(* IEC 61131-3 sources: F100R_S278_Temperville/MyController.device.xml.v3^/Plc Logic.plclogic.xml.v3^/Application.application.xml.v3^/04_PID/HEAT/10_Temperatura (part 3) *)

//// SUPERIORES

// Controle Resistencia 51

SR_ControleTemperatura.FbCrtlAquecimento[51](
	i_xEnable:= InterfaceHeat.P_xHabTemp51 OR xLigaDesligaSupG01,
	i_rSetPoint:= rSetPointTemperaturaSuperior[1],
	i_rProcessValue:= I_rTemperatura51,
	i_xManualMode:= ,
	i_rManualValue:= ,
	i_xAutoTune:= TEMP.xAutoTuneTemp51 OR xAutoTuneTempGeral,
	i_xHold:= ,
	i_xReset:= InterfaceHeat.xReset,
	i_stTemperatureControl:= stTemperatureControl[51],
	iq_etSelectParameterSetPID:= etSelectParameterSetPID[51],
	iq_stParameterSetsPID:= stParameterSetsPID[51],
	q_xActive=> ,
	q_xReady=> ,
	q_xError=> TEMP.xCrtlTemperatura[51],
	q_etResult=> TEMP.iCrtlTempStsTemp51,
	q_sResultMsg=> ,
	q_rAnalogOutput=> TEMP.rCrtlTempPotTemp51,
	q_xPwmOutput=> Q_xAquecimento51,
	q_xAutoTuneActive=> TEMP.xAutoTuneAtivoTemp51,
	q_etStatusAutoTune=> TEMP.iAutoTuneStsTemp51);

rPwmEntrada[51]:= TEMP.rCrtlTempPotTemp51*(rSetPorcentagemSuperior[1]/100);

PWM[51].i_stPara.tCyclTime:=T#10MS;
PWM[51].i_stPara.tPwmPeriod:=T#1000MS;
PWM[51](
	i_xEn:= 	xHabilitaBlocosControleSuperior,
	i_rIput:= 	rPwmEntrada[51],
	i_stPara:= 	,
	i_xErrRst:= xResetPid,
	q_xEn=> 	,
	q_xBusy=> 	,
	q_xPstv=> 	Q_xAquecimentoPwm51,
	q_xNgtv=> 	,
	q_xErr=> 	,
	q_uiErrId=> );

// Controle Resistencia 52

SR_ControleTemperatura.FbCrtlAquecimento[52](
	i_xEnable:= InterfaceHeat.P_xHabTemp52 OR xLigaDesligaSupG02,
	i_rSetPoint:= rSetPointTemperaturaSuperior[2],
	i_rProcessValue:= I_rTemperatura52,
	i_xManualMode:= ,
	i_rManualValue:= ,
	i_xAutoTune:= TEMP.xAutoTuneTemp52 OR xAutoTuneTempGeral,
	i_xHold:= ,
	i_xReset:= InterfaceHeat.xReset,
	i_stTemperatureControl:= stTemperatureControl[52],
	iq_etSelectParameterSetPID:= etSelectParameterSetPID[52],
	iq_stParameterSetsPID:= stParameterSetsPID[52],
	q_xActive=> ,
	q_xReady=> ,
	q_xError=> TEMP.xCrtlTemperatura[52],
	q_etResult=> TEMP.iCrtlTempStsTemp52,
	q_sResultMsg=> ,
	q_rAnalogOutput=> TEMP.rCrtlTempPotTemp52,
	q_xPwmOutput=> Q_xAquecimento52,
	q_xAutoTuneActive=> TEMP.xAutoTuneAtivoTemp52,
	q_etStatusAutoTune=> TEMP.iAutoTuneStsTemp52);

rPwmEntrada[52]:= TEMP.rCrtlTempPotTemp52*(rSetPorcentagemSuperior[2]/100);

PWM[52].i_stPara.tCyclTime:=T#10MS;
PWM[52].i_stPara.tPwmPeriod:=T#1000MS;
PWM[52](
	i_xEn:= 	xHabilitaBlocosControleSuperior,
	i_rIput:= 	rPwmEntrada[52],
	i_stPara:= 	,
	i_xErrRst:= xResetPid,
	q_xEn=> 	,
	q_xBusy=> 	,
	q_xPstv=> 	Q_xAquecimentoPwm52,
	q_xNgtv=> 	,
	q_xErr=> 	,
	q_uiErrId=> );

// Controle Resistencia 53

SR_ControleTemperatura.FbCrtlAquecimento[53](
	i_xEnable:= InterfaceHeat.P_xHabTemp53 OR xLigaDesligaSupG01,
	i_rSetPoint:= rSetPointTemperaturaSuperior[3],
	i_rProcessValue:= I_rTemperatura53,
	i_xManualMode:= ,
	i_rManualValue:= ,
	i_xAutoTune:= TEMP.xAutoTuneTemp53 OR xAutoTuneTempGeral,
	i_xHold:= ,
	i_xReset:= InterfaceHeat.xReset,
	i_stTemperatureControl:= stTemperatureControl[53],
	iq_etSelectParameterSetPID:= etSelectParameterSetPID[53],
	iq_stParameterSetsPID:= stParameterSetsPID[53],
	q_xActive=> ,
	q_xReady=> ,
	q_xError=> TEMP.xCrtlTemperatura[53],
	q_etResult=> TEMP.iCrtlTempStsTemp53,
	q_sResultMsg=> ,
	q_rAnalogOutput=> TEMP.rCrtlTempPotTemp53,
	q_xPwmOutput=> Q_xAquecimento53,
	q_xAutoTuneActive=> TEMP.xAutoTuneAtivoTemp53,
	q_etStatusAutoTune=> TEMP.iAutoTuneStsTemp53);

rPwmEntrada[53]:= TEMP.rCrtlTempPotTemp53*(rSetPorcentagemSuperior[3]/100);

PWM[53].i_stPara.tCyclTime:=T#10MS;
PWM[53].i_stPara.tPwmPeriod:=T#1000MS;
PWM[53](
	i_xEn:= 	xHabilitaBlocosControleSuperior,
	i_rIput:= 	rPwmEntrada[53],
	i_stPara:= 	,
	i_xErrRst:= xResetPid,
	q_xEn=> 	,
	q_xBusy=> 	,
	q_xPstv=> 	Q_xAquecimentoPwm53,
	q_xNgtv=> 	,
	q_xErr=> 	,
	q_uiErrId=> );

// Controle Resistencia 54

SR_ControleTemperatura.FbCrtlAquecimento[54](
	i_xEnable:= InterfaceHeat.P_xHabTemp54 OR xLigaDesligaSupG02,
	i_rSetPoint:= rSetPointTemperaturaSuperior[4],
	i_rProcessValue:= I_rTemperatura54,
	i_xManualMode:= ,
	i_rManualValue:= ,
	i_xAutoTune:= TEMP.xAutoTuneTemp54 OR xAutoTuneTempGeral,
	i_xHold:= ,
	i_xReset:= InterfaceHeat.xReset,
	i_stTemperatureControl:= stTemperatureControl[54],
	iq_etSelectParameterSetPID:= etSelectParameterSetPID[54],
	iq_stParameterSetsPID:= stParameterSetsPID[54],
	q_xActive=> ,
	q_xReady=> ,
	q_xError=> TEMP.xCrtlTemperatura[54],
	q_etResult=> TEMP.iCrtlTempStsTemp54,
	q_sResultMsg=> ,
	q_rAnalogOutput=> TEMP.rCrtlTempPotTemp54,
	q_xPwmOutput=> Q_xAquecimento54,
	q_xAutoTuneActive=> TEMP.xAutoTuneAtivoTemp54,
	q_etStatusAutoTune=> TEMP.iAutoTuneStsTemp54);

rPwmEntrada[54]:= TEMP.rCrtlTempPotTemp54*(rSetPorcentagemSuperior[4]/100);

PWM[54].i_stPara.tCyclTime:=T#10MS;
PWM[54].i_stPara.tPwmPeriod:=T#1000MS;
PWM[54](
	i_xEn:= 	xHabilitaBlocosControleSuperior,
	i_rIput:= 	rPwmEntrada[54],
	i_stPara:= 	,
	i_xErrRst:= xResetPid,
	q_xEn=> 	,
	q_xBusy=> 	,
	q_xPstv=> 	Q_xAquecimentoPwm54,
	q_xNgtv=> 	,
	q_xErr=> 	,
	q_uiErrId=> );

// Controle Resistencia 55

SR_ControleTemperatura.FbCrtlAquecimento[55](
	i_xEnable:= InterfaceHeat.P_xHabTemp55 OR xLigaDesligaSupG01,
	i_rSetPoint:= rSetPointTemperaturaSuperior[5],
	i_rProcessValue:= I_rTemperatura55,
	i_xManualMode:= ,
	i_rManualValue:= ,
	i_xAutoTune:= TEMP.xAutoTuneTemp55 OR xAutoTuneTempGeral,
	i_xHold:= ,
	i_xReset:= InterfaceHeat.xReset,
	i_stTemperatureControl:= stTemperatureControl[55],
	iq_etSelectParameterSetPID:= etSelectParameterSetPID[55],
	iq_stParameterSetsPID:= stParameterSetsPID[55],
	q_xActive=> ,
	q_xReady=> ,
	q_xError=> TEMP.xCrtlTemperatura[55],
	q_etResult=> TEMP.iCrtlTempStsTemp55,
	q_sResultMsg=> ,
	q_rAnalogOutput=> TEMP.rCrtlTempPotTemp55,
	q_xPwmOutput=> Q_xAquecimento55,
	q_xAutoTuneActive=> TEMP.xAutoTuneAtivoTemp55,
	q_etStatusAutoTune=> TEMP.iAutoTuneStsTemp55);

rPwmEntrada[55]:= TEMP.rCrtlTempPotTemp55*(rSetPorcentagemSuperior[5]/100);

PWM[55].i_stPara.tCyclTime:=T#10MS;
PWM[55].i_stPara.tPwmPeriod:=T#1000MS;
PWM[55](
	i_xEn:= 	xHabilitaBlocosControleSuperior,
	i_rIput:= 	rPwmEntrada[55],
	i_stPara:= 	,
	i_xErrRst:= xResetPid,
	q_xEn=> 	,
	q_xBusy=> 	,
	q_xPstv=> 	Q_xAquecimentoPwm55,
	q_xNgtv=> 	,
	q_xErr=> 	,
	q_uiErrId=> );

// Controle Resistencia 56

SR_ControleTemperatura.FbCrtlAquecimento[56](
	i_xEnable:= InterfaceHeat.P_xHabTemp56 OR xLigaDesligaSupG02,
	i_rSetPoint:= rSetPointTemperaturaSuperior[6],
	i_rProcessValue:= I_rTemperatura56,
	i_xManualMode:= ,
	i_rManualValue:= ,
	i_xAutoTune:= TEMP.xAutoTuneTemp56 OR xAutoTuneTempGeral,
	i_xHold:= ,
	i_xReset:= InterfaceHeat.xReset,
	i_stTemperatureControl:= stTemperatureControl[56],
	iq_etSelectParameterSetPID:= etSelectParameterSetPID[56],
	iq_stParameterSetsPID:= stParameterSetsPID[56],
	q_xActive=> ,
	q_xReady=> ,
	q_xError=> TEMP.xCrtlTemperatura[56],
	q_etResult=> TEMP.iCrtlTempStsTemp56,
	q_sResultMsg=> ,
	q_rAnalogOutput=> TEMP.rCrtlTempPotTemp56,
	q_xPwmOutput=> Q_xAquecimento56,
	q_xAutoTuneActive=> TEMP.xAutoTuneAtivoTemp56,
	q_etStatusAutoTune=> TEMP.iAutoTuneStsTemp56);

rPwmEntrada[56]:= TEMP.rCrtlTempPotTemp56*(rSetPorcentagemSuperior[6]/100);

PWM[56].i_stPara.tCyclTime:=T#10MS;
PWM[56].i_stPara.tPwmPeriod:=T#1000MS;
PWM[56](
	i_xEn:= 	xHabilitaBlocosControleSuperior,
	i_rIput:= 	rPwmEntrada[56],
	i_stPara:= 	,
	i_xErrRst:= xResetPid,
	q_xEn=> 	,
	q_xBusy=> 	,
	q_xPstv=> 	Q_xAquecimentoPwm56,
	q_xNgtv=> 	,
	q_xErr=> 	,
	q_uiErrId=> );

// Controle Resistencia 57

SR_ControleTemperatura.FbCrtlAquecimento[57](
	i_xEnable:= InterfaceHeat.P_xHabTemp57 OR xLigaDesligaSupG01,
	i_rSetPoint:= rSetPointTemperaturaSuperior[7],
	i_rProcessValue:= I_rTemperatura57,
	i_xManualMode:= ,
	i_rManualValue:= ,
	i_xAutoTune:= TEMP.xAutoTuneTemp57 OR xAutoTuneTempGeral,
	i_xHold:= ,
	i_xReset:= InterfaceHeat.xReset,
	i_stTemperatureControl:= stTemperatureControl[57],
	iq_etSelectParameterSetPID:= etSelectParameterSetPID[57],
	iq_stParameterSetsPID:= stParameterSetsPID[57],
	q_xActive=> ,
	q_xReady=> ,
	q_xError=> TEMP.xCrtlTemperatura[57],
	q_etResult=> TEMP.iCrtlTempStsTemp57,
	q_sResultMsg=> ,
	q_rAnalogOutput=> TEMP.rCrtlTempPotTemp57,
	q_xPwmOutput=> Q_xAquecimento57,
	q_xAutoTuneActive=> TEMP.xAutoTuneAtivoTemp57,
	q_etStatusAutoTune=> TEMP.iAutoTuneStsTemp57);

rPwmEntrada[57]:= TEMP.rCrtlTempPotTemp57*(rSetPorcentagemSuperior[7]/100);

PWM[57].i_stPara.tCyclTime:=T#10MS;
PWM[57].i_stPara.tPwmPeriod:=T#1000MS;
PWM[57](
	i_xEn:= 	xHabilitaBlocosControleSuperior,
	i_rIput:= 	rPwmEntrada[57],
	i_stPara:= 	,
	i_xErrRst:= xResetPid,
	q_xEn=> 	,
	q_xBusy=> 	,
	q_xPstv=> 	Q_xAquecimentoPwm57,
	q_xNgtv=> 	,
	q_xErr=> 	,
	q_uiErrId=> );

	// Controle Resistencia 58

SR_ControleTemperatura.FbCrtlAquecimento[58](
	i_xEnable:= InterfaceHeat.P_xHabTemp58 OR xLigaDesligaSupG02,
	i_rSetPoint:= rSetPointTemperaturaSuperior[8],
	i_rProcessValue:= I_rTemperatura58,
	i_xManualMode:= ,
	i_rManualValue:= ,
	i_xAutoTune:= TEMP.xAutoTuneTemp58 OR xAutoTuneTempGeral,
	i_xHold:= ,
	i_xReset:= InterfaceHeat.xReset,
	i_stTemperatureControl:= stTemperatureControl[58],
	iq_etSelectParameterSetPID:= etSelectParameterSetPID[58],
	iq_stParameterSetsPID:= stParameterSetsPID[58],
	q_xActive=> ,
	q_xReady=> ,
	q_xError=> TEMP.xCrtlTemperatura[58],
	q_etResult=> TEMP.iCrtlTempStsTemp58,
	q_sResultMsg=> ,
	q_rAnalogOutput=> TEMP.rCrtlTempPotTemp58,
	q_xPwmOutput=> Q_xAquecimento58,
	q_xAutoTuneActive=> TEMP.xAutoTuneAtivoTemp58,
	q_etStatusAutoTune=> TEMP.iAutoTuneStsTemp58);

rPwmEntrada[58]:= TEMP.rCrtlTempPotTemp58*(rSetPorcentagemSuperior[8]/100);

PWM[58].i_stPara.tCyclTime:=T#10MS;
PWM[58].i_stPara.tPwmPeriod:=T#1000MS;
PWM[58](
	i_xEn:= 	xHabilitaBlocosControleSuperior,
	i_rIput:= 	rPwmEntrada[58],
	i_stPara:= 	,
	i_xErrRst:= xResetPid,
	q_xEn=> 	,
	q_xBusy=> 	,
	q_xPstv=> 	Q_xAquecimentoPwm58,
	q_xNgtv=> 	,
	q_xErr=> 	,
	q_uiErrId=> );

	// Controle Resistencia 59

SR_ControleTemperatura.FbCrtlAquecimento[59](
	i_xEnable:= InterfaceHeat.P_xHabTemp59 OR xLigaDesligaSupG01,
	i_rSetPoint:= rSetPointTemperaturaSuperior[9],
	i_rProcessValue:= I_rTemperatura59,
	i_xManualMode:= ,
	i_rManualValue:= ,
	i_xAutoTune:= TEMP.xAutoTuneTemp59 OR xAutoTuneTempGeral,
	i_xHold:= ,
	i_xReset:= InterfaceHeat.xReset,
	i_stTemperatureControl:= stTemperatureControl[59],
	iq_etSelectParameterSetPID:= etSelectParameterSetPID[59],
	iq_stParameterSetsPID:= stParameterSetsPID[59],
	q_xActive=> ,
	q_xReady=> ,
	q_xError=> TEMP.xCrtlTemperatura[59],
	q_etResult=> TEMP.iCrtlTempStsTemp59,
	q_sResultMsg=> ,
	q_rAnalogOutput=> TEMP.rCrtlTempPotTemp59,
	q_xPwmOutput=> Q_xAquecimento59,
	q_xAutoTuneActive=> TEMP.xAutoTuneAtivoTemp59,
	q_etStatusAutoTune=> TEMP.iAutoTuneStsTemp59);

rPwmEntrada[59]:= TEMP.rCrtlTempPotTemp59*(rSetPorcentagemSuperior[9]/100);

PWM[59].i_stPara.tCyclTime:=T#10MS;
PWM[59].i_stPara.tPwmPeriod:=T#1000MS;
PWM[59](
	i_xEn:= 	xHabilitaBlocosControleSuperior,
	i_rIput:= 	rPwmEntrada[59],
	i_stPara:= 	,
	i_xErrRst:= xResetPid,
	q_xEn=> 	,
	q_xBusy=> 	,
	q_xPstv=> 	Q_xAquecimentoPwm59,
	q_xNgtv=> 	,
	q_xErr=> 	,
	q_uiErrId=> );

	// Controle Resistencia 60

SR_ControleTemperatura.FbCrtlAquecimento[60](
	i_xEnable:= InterfaceHeat.P_xHabTemp60 OR xLigaDesligaSupG02,
	i_rSetPoint:= rSetPointTemperaturaSuperior[10],
	i_rProcessValue:= I_rTemperatura60,
	i_xManualMode:= ,
	i_rManualValue:= ,
	i_xAutoTune:= TEMP.xAutoTuneTemp60 OR xAutoTuneTempGeral,
	i_xHold:= ,
	i_xReset:= InterfaceHeat.xReset,
	i_stTemperatureControl:= stTemperatureControl[60],
	iq_etSelectParameterSetPID:= etSelectParameterSetPID[60],
	iq_stParameterSetsPID:= stParameterSetsPID[60],
	q_xActive=> ,
	q_xReady=> ,
	q_xError=> TEMP.xCrtlTemperatura[60],
	q_etResult=> TEMP.iCrtlTempStsTemp60,
	q_sResultMsg=> ,
	q_rAnalogOutput=> TEMP.rCrtlTempPotTemp60,
	q_xPwmOutput=> Q_xAquecimento60,
	q_xAutoTuneActive=> TEMP.xAutoTuneAtivoTemp60,
	q_etStatusAutoTune=> TEMP.iAutoTuneStsTemp60);

rPwmEntrada[60]:= TEMP.rCrtlTempPotTemp60*(rSetPorcentagemSuperior[10]/100);

PWM[60].i_stPara.tCyclTime:=T#10MS;
PWM[60].i_stPara.tPwmPeriod:=T#1000MS;
PWM[60](
	i_xEn:= 	xHabilitaBlocosControleSuperior,
	i_rIput:= 	rPwmEntrada[60],
	i_stPara:= 	,
	i_xErrRst:= xResetPid,
	q_xEn=> 	,
	q_xBusy=> 	,
	q_xPstv=> 	Q_xAquecimentoPwm60,
	q_xNgtv=> 	,
	q_xErr=> 	,
	q_uiErrId=> );

// Controle Resistencia 61

SR_ControleTemperatura.FbCrtlAquecimento[61](
	i_xEnable:= InterfaceHeat.P_xHabTemp61 OR xLigaDesligaSupG02,
	i_rSetPoint:= rSetPointTemperaturaSuperior[11],
	i_rProcessValue:= I_rTemperatura61,
	i_xManualMode:= ,
	i_rManualValue:= ,
	i_xAutoTune:= TEMP.xAutoTuneTemp61 OR xAutoTuneTempGeral,
	i_xHold:= ,
	i_xReset:= InterfaceHeat.xReset,
	i_stTemperatureControl:= stTemperatureControl[61],
	iq_etSelectParameterSetPID:= etSelectParameterSetPID[61],
	iq_stParameterSetsPID:= stParameterSetsPID[61],
	q_xActive=> ,
	q_xReady=> ,
	q_xError=> TEMP.xCrtlTemperatura[61],
	q_etResult=> TEMP.iCrtlTempStsTemp61,
	q_sResultMsg=> ,
	q_rAnalogOutput=> TEMP.rCrtlTempPotTemp61,
	q_xPwmOutput=> Q_xAquecimento61,
	q_xAutoTuneActive=> TEMP.xAutoTuneAtivoTemp61,
	q_etStatusAutoTune=> TEMP.iAutoTuneStsTemp61);

rPwmEntrada[61]:= TEMP.rCrtlTempPotTemp6*(rSetPorcentagemSuperior[11]/100);

PWM[61].i_stPara.tCyclTime:=T#10MS;
PWM[61].i_stPara.tPwmPeriod:=T#1000MS;
PWM[61](
	i_xEn:= 	xHabilitaBlocosControleSuperior,
	i_rIput:= 	rPwmEntrada[61],
	i_stPara:= 	,
	i_xErrRst:= xResetPid,
	q_xEn=> 	,
	q_xBusy=> 	,
	q_xPstv=> 	Q_xAquecimentoPwm61,
	q_xNgtv=> 	,
	q_xErr=> 	,
	q_uiErrId=> );

// Controle Resistencia 62

SR_ControleTemperatura.FbCrtlAquecimento[62](
	i_xEnable:= InterfaceHeat.P_xHabTemp62 OR xLigaDesligaSupG01,
	i_rSetPoint:= rSetPointTemperaturaSuperior[12],
	i_rProcessValue:= I_rTemperatura62,
	i_xManualMode:= ,
	i_rManualValue:= ,
	i_xAutoTune:= TEMP.xAutoTuneTemp62 OR xAutoTuneTempGeral,
	i_xHold:= ,
	i_xReset:= InterfaceHeat.xReset,
	i_stTemperatureControl:= stTemperatureControl[62],
	iq_etSelectParameterSetPID:= etSelectParameterSetPID[62],
	iq_stParameterSetsPID:= stParameterSetsPID[62],
	q_xActive=> ,
	q_xReady=> ,
	q_xError=> TEMP.xCrtlTemperatura[62],
	q_etResult=> TEMP.iCrtlTempStsTemp62,
	q_sResultMsg=> ,
	q_rAnalogOutput=> TEMP.rCrtlTempPotTemp62,
	q_xPwmOutput=> Q_xAquecimento62,
	q_xAutoTuneActive=> TEMP.xAutoTuneAtivoTemp62,
	q_etStatusAutoTune=> TEMP.iAutoTuneStsTemp62);

rPwmEntrada[62]:= TEMP.rCrtlTempPotTemp62*(rSetPorcentagemSuperior[12]/100);

PWM[62].i_stPara.tCyclTime:=T#10MS;
PWM[62].i_stPara.tPwmPeriod:=T#1000MS;
PWM[62](
	i_xEn:= 	xHabilitaBlocosControleSuperior,
	i_rIput:= 	rPwmEntrada[62],
	i_stPara:= 	,
	i_xErrRst:= xResetPid,
	q_xEn=> 	,
	q_xBusy=> 	,
	q_xPstv=> 	Q_xAquecimentoPwm62,
	q_xNgtv=> 	,
	q_xErr=> 	,
	q_uiErrId=> );

// Controle Resistencia 63

SR_ControleTemperatura.FbCrtlAquecimento[63](
	i_xEnable:= InterfaceHeat.P_xHabTemp63 OR xLigaDesligaSupG02,
	i_rSetPoint:= rSetPointTemperaturaSuperior[13],
	i_rProcessValue:= I_rTemperatura63,
	i_xManualMode:= ,
	i_rManualValue:= ,
	i_xAutoTune:= TEMP.xAutoTuneTemp63 OR xAutoTuneTempGeral,
	i_xHold:= ,
	i_xReset:= InterfaceHeat.xReset,
	i_stTemperatureControl:= stTemperatureControl[63],
	iq_etSelectParameterSetPID:= etSelectParameterSetPID[63],
	iq_stParameterSetsPID:= stParameterSetsPID[63],
	q_xActive=> ,
	q_xReady=> ,
	q_xError=> TEMP.xCrtlTemperatura[63],
	q_etResult=> TEMP.iCrtlTempStsTemp63,
	q_sResultMsg=> ,
	q_rAnalogOutput=> TEMP.rCrtlTempPotTemp63,
	q_xPwmOutput=> Q_xAquecimento63,
	q_xAutoTuneActive=> TEMP.xAutoTuneAtivoTemp63,
	q_etStatusAutoTune=> TEMP.iAutoTuneStsTemp63);

rPwmEntrada[63]:= TEMP.rCrtlTempPotTemp63*(rSetPorcentagemSuperior[13]/100);

PWM[63].i_stPara.tCyclTime:=T#10MS;
PWM[63].i_stPara.tPwmPeriod:=T#1000MS;
PWM[63](
	i_xEn:= 	xHabilitaBlocosControleSuperior,
	i_rIput:= 	rPwmEntrada[63],
	i_stPara:= 	,
	i_xErrRst:= xResetPid,
	q_xEn=> 	,
	q_xBusy=> 	,
	q_xPstv=> 	Q_xAquecimentoPwm63,
	q_xNgtv=> 	,
	q_xErr=> 	,
	q_uiErrId=> );

// Controle Resistencia 64

SR_ControleTemperatura.FbCrtlAquecimento[64](
	i_xEnable:= InterfaceHeat.P_xHabTemp64 OR xLigaDesligaSupG01,
	i_rSetPoint:= rSetPointTemperaturaSuperior[14],
	i_rProcessValue:= I_rTemperatura64,
	i_xManualMode:= ,
	i_rManualValue:= ,
	i_xAutoTune:= TEMP.xAutoTuneTemp64 OR xAutoTuneTempGeral,
	i_xHold:= ,
	i_xReset:= InterfaceHeat.xReset,
	i_stTemperatureControl:= stTemperatureControl[64],
	iq_etSelectParameterSetPID:= etSelectParameterSetPID[64],
	iq_stParameterSetsPID:= stParameterSetsPID[64],
	q_xActive=> ,
	q_xReady=> ,
	q_xError=> TEMP.xCrtlTemperatura[64],
	q_etResult=> TEMP.iCrtlTempStsTemp64,
	q_sResultMsg=> ,
	q_rAnalogOutput=> TEMP.rCrtlTempPotTemp64,
	q_xPwmOutput=> Q_xAquecimento64,
	q_xAutoTuneActive=> TEMP.xAutoTuneAtivoTemp64,
	q_etStatusAutoTune=> TEMP.iAutoTuneStsTemp64);

rPwmEntrada[64]:= TEMP.rCrtlTempPotTemp64*(rSetPorcentagemSuperior[14]/100);

PWM[64].i_stPara.tCyclTime:=T#10MS;
PWM[64].i_stPara.tPwmPeriod:=T#1000MS;
PWM[64](
	i_xEn:= 	xHabilitaBlocosControleSuperior,
	i_rIput:= 	rPwmEntrada[64],
	i_stPara:= 	,
	i_xErrRst:= xResetPid,
	q_xEn=> 	,
	q_xBusy=> 	,
	q_xPstv=> 	Q_xAquecimentoPwm64,
	q_xNgtv=> 	,
	q_xErr=> 	,
	q_uiErrId=> );

// Controle Resistencia 65

SR_ControleTemperatura.FbCrtlAquecimento[65](
	i_xEnable:= InterfaceHeat.P_xHabTemp65 OR xLigaDesligaSupG02,
	i_rSetPoint:= rSetPointTemperaturaSuperior[15],
	i_rProcessValue:= I_rTemperatura65,
	i_xManualMode:= ,
	i_rManualValue:= ,
	i_xAutoTune:= TEMP.xAutoTuneTemp65 OR xAutoTuneTempGeral,
	i_xHold:= ,
	i_xReset:= InterfaceHeat.xReset,
	i_stTemperatureControl:= stTemperatureControl[65],
	iq_etSelectParameterSetPID:= etSelectParameterSetPID[65],
	iq_stParameterSetsPID:= stParameterSetsPID[65],
	q_xActive=> ,
	q_xReady=> ,
	q_xError=> TEMP.xCrtlTemperatura[65],
	q_etResult=> TEMP.iCrtlTempStsTemp65,
	q_sResultMsg=> ,
	q_rAnalogOutput=> TEMP.rCrtlTempPotTemp65,
	q_xPwmOutput=> Q_xAquecimento65,
	q_xAutoTuneActive=> TEMP.xAutoTuneAtivoTemp65,
	q_etStatusAutoTune=> TEMP.iAutoTuneStsTemp65);

rPwmEntrada[65]:= TEMP.rCrtlTempPotTemp65*(rSetPorcentagemSuperior[15]/100);

PWM[65].i_stPara.tCyclTime:=T#10MS;
PWM[65].i_stPara.tPwmPeriod:=T#1000MS;
PWM[65](
	i_xEn:= 	xHabilitaBlocosControleSuperior,
	i_rIput:= 	rPwmEntrada[65],
	i_stPara:= 	,
	i_xErrRst:= xResetPid,
	q_xEn=> 	,
	q_xBusy=> 	,
	q_xPstv=> 	Q_xAquecimentoPwm65,
	q_xNgtv=> 	,
	q_xErr=> 	,
	q_uiErrId=> );

// Controle Resistencia 66

SR_ControleTemperatura.FbCrtlAquecimento[66](
	i_xEnable:= InterfaceHeat.P_xHabTemp66 OR xLigaDesligaSupG01,
	i_rSetPoint:= rSetPointTemperaturaSuperior[16],
	i_rProcessValue:= I_rTemperatura66,
	i_xManualMode:= ,
	i_rManualValue:= ,
	i_xAutoTune:= TEMP.xAutoTuneTemp66 OR xAutoTuneTempGeral,
	i_xHold:= ,
	i_xReset:= InterfaceHeat.xReset,
	i_stTemperatureControl:= stTemperatureControl[66],
	iq_etSelectParameterSetPID:= etSelectParameterSetPID[66],
	iq_stParameterSetsPID:= stParameterSetsPID[66],
	q_xActive=> ,
	q_xReady=> ,
	q_xError=> TEMP.xCrtlTemperatura[66],
	q_etResult=> TEMP.iCrtlTempStsTemp66,
	q_sResultMsg=> ,
	q_rAnalogOutput=> TEMP.rCrtlTempPotTemp66,
	q_xPwmOutput=> Q_xAquecimento66,
	q_xAutoTuneActive=> TEMP.xAutoTuneAtivoTemp66,
	q_etStatusAutoTune=> TEMP.iAutoTuneStsTemp66);

rPwmEntrada[66]:= TEMP.rCrtlTempPotTemp66*(rSetPorcentagemSuperior[16]/100);

PWM[66].i_stPara.tCyclTime:=T#10MS;
PWM[66].i_stPara.tPwmPeriod:=T#1000MS;
PWM[66](
	i_xEn:= 	xHabilitaBlocosControleSuperior,
	i_rIput:= 	rPwmEntrada[66],
	i_stPara:= 	,
	i_xErrRst:= xResetPid,
	q_xEn=> 	,
	q_xBusy=> 	,
	q_xPstv=> 	Q_xAquecimentoPwm66,
	q_xNgtv=> 	,
	q_xErr=> 	,
	q_uiErrId=> );

// Controle Resistencia 67

SR_ControleTemperatura.FbCrtlAquecimento[67](
	i_xEnable:= InterfaceHeat.P_xHabTemp67 OR xLigaDesligaSupG02,
	i_rSetPoint:= rSetPointTemperaturaSuperior[17],
	i_rProcessValue:= I_rTemperatura67,
	i_xManualMode:= ,
	i_rManualValue:= ,
	i_xAutoTune:= TEMP.xAutoTuneTemp67 OR xAutoTuneTempGeral,
	i_xHold:= ,
	i_xReset:= InterfaceHeat.xReset,
	i_stTemperatureControl:= stTemperatureControl[67],
	iq_etSelectParameterSetPID:= etSelectParameterSetPID[67],
	iq_stParameterSetsPID:= stParameterSetsPID[67],
	q_xActive=> ,
	q_xReady=> ,
	q_xError=> TEMP.xCrtlTemperatura[67],
	q_etResult=> TEMP.iCrtlTempStsTemp67,
	q_sResultMsg=> ,
	q_rAnalogOutput=> TEMP.rCrtlTempPotTemp67,
	q_xPwmOutput=> Q_xAquecimento67,
	q_xAutoTuneActive=> TEMP.xAutoTuneAtivoTemp67,
	q_etStatusAutoTune=> TEMP.iAutoTuneStsTemp67);

rPwmEntrada[67]:= TEMP.rCrtlTempPotTemp67*(rSetPorcentagemSuperior[17]/100);

PWM[67].i_stPara.tCyclTime:=T#10MS;
PWM[67].i_stPara.tPwmPeriod:=T#1000MS;
PWM[67](
	i_xEn:= 	xHabilitaBlocosControleSuperior,
	i_rIput:= 	rPwmEntrada[67],
	i_stPara:= 	,
	i_xErrRst:= xResetPid,
	q_xEn=> 	,
	q_xBusy=> 	,
	q_xPstv=> 	Q_xAquecimentoPwm67,
	q_xNgtv=> 	,
	q_xErr=> 	,
	q_uiErrId=> );

	// Controle Resistencia 68

SR_ControleTemperatura.FbCrtlAquecimento[68](
	i_xEnable:= InterfaceHeat.P_xHabTemp68 OR xLigaDesligaSupG01,
	i_rSetPoint:= rSetPointTemperaturaSuperior[18],
	i_rProcessValue:= I_rTemperatura68,
	i_xManualMode:= ,
	i_rManualValue:= ,
	i_xAutoTune:= TEMP.xAutoTuneTemp68 OR xAutoTuneTempGeral,
	i_xHold:= ,
	i_xReset:= InterfaceHeat.xReset,
	i_stTemperatureControl:= stTemperatureControl[68],
	iq_etSelectParameterSetPID:= etSelectParameterSetPID[68],
	iq_stParameterSetsPID:= stParameterSetsPID[68],
	q_xActive=> ,
	q_xReady=> ,
	q_xError=> TEMP.xCrtlTemperatura[68],
	q_etResult=> TEMP.iCrtlTempStsTemp68,
	q_sResultMsg=> ,
	q_rAnalogOutput=> TEMP.rCrtlTempPotTemp68,
	q_xPwmOutput=> Q_xAquecimento68,
	q_xAutoTuneActive=> TEMP.xAutoTuneAtivoTemp68,
	q_etStatusAutoTune=> TEMP.iAutoTuneStsTemp68);

rPwmEntrada[68]:= TEMP.rCrtlTempPotTemp68*(rSetPorcentagemSuperior[18]/100);

PWM[68].i_stPara.tCyclTime:=T#10MS;
PWM[68].i_stPara.tPwmPeriod:=T#1000MS;
PWM[68](
	i_xEn:= 	xHabilitaBlocosControleSuperior,
	i_rIput:= 	rPwmEntrada[68],
	i_stPara:= 	,
	i_xErrRst:= xResetPid,
	q_xEn=> 	,
	q_xBusy=> 	,
	q_xPstv=> 	Q_xAquecimentoPwm68,
	q_xNgtv=> 	,
	q_xErr=> 	,
	q_uiErrId=> );

	// Controle Resistencia 69

SR_ControleTemperatura.FbCrtlAquecimento[69](
	i_xEnable:= InterfaceHeat.P_xHabTemp69 OR xLigaDesligaSupG02,
	i_rSetPoint:= rSetPointTemperaturaSuperior[19],
	i_rProcessValue:= I_rTemperatura69,
	i_xManualMode:= ,
	i_rManualValue:= ,
	i_xAutoTune:= TEMP.xAutoTuneTemp69 OR xAutoTuneTempGeral,
	i_xHold:= ,
	i_xReset:= InterfaceHeat.xReset,
	i_stTemperatureControl:= stTemperatureControl[69],
	iq_etSelectParameterSetPID:= etSelectParameterSetPID[69],
	iq_stParameterSetsPID:= stParameterSetsPID[69],
	q_xActive=> ,
	q_xReady=> ,
	q_xError=> TEMP.xCrtlTemperatura[69],
	q_etResult=> TEMP.iCrtlTempStsTemp69,
	q_sResultMsg=> ,
	q_rAnalogOutput=> TEMP.rCrtlTempPotTemp69,
	q_xPwmOutput=> Q_xAquecimento69,
	q_xAutoTuneActive=> TEMP.xAutoTuneAtivoTemp69,
	q_etStatusAutoTune=> TEMP.iAutoTuneStsTemp69);

rPwmEntrada[69]:= TEMP.rCrtlTempPotTemp69*(rSetPorcentagemSuperior[19]/100);

PWM[69].i_stPara.tCyclTime:=T#10MS;
PWM[69].i_stPara.tPwmPeriod:=T#1000MS;
PWM[69](
	i_xEn:= 	xHabilitaBlocosControleSuperior,
	i_rIput:= 	rPwmEntrada[69],
	i_stPara:= 	,
	i_xErrRst:= xResetPid,
	q_xEn=> 	,
	q_xBusy=> 	,
	q_xPstv=> 	Q_xAquecimentoPwm69,
	q_xNgtv=> 	,
	q_xErr=> 	,
	q_uiErrId=> );

	// Controle Resistencia 70

SR_ControleTemperatura.FbCrtlAquecimento[70](
	i_xEnable:= InterfaceHeat.P_xHabTemp70 OR xLigaDesligaSupG01,
	i_rSetPoint:= rSetPointTemperaturaSuperior[20],
	i_rProcessValue:= I_rTemperatura70,
	i_xManualMode:= ,
	i_rManualValue:= ,
	i_xAutoTune:= TEMP.xAutoTuneTemp70 OR xAutoTuneTempGeral,
	i_xHold:= ,
	i_xReset:= InterfaceHeat.xReset,
	i_stTemperatureControl:= stTemperatureControl[70],
	iq_etSelectParameterSetPID:= etSelectParameterSetPID[70],
	iq_stParameterSetsPID:= stParameterSetsPID[70],
	q_xActive=> ,
	q_xReady=> ,
	q_xError=> TEMP.xCrtlTemperatura[70],
	q_etResult=> TEMP.iCrtlTempStsTemp70,
	q_sResultMsg=> ,
	q_rAnalogOutput=> TEMP.rCrtlTempPotTemp70,
	q_xPwmOutput=> Q_xAquecimento70,
	q_xAutoTuneActive=> TEMP.xAutoTuneAtivoTemp70,
	q_etStatusAutoTune=> TEMP.iAutoTuneStsTemp70);

rPwmEntrada[70]:= TEMP.rCrtlTempPotTemp70*(rSetPorcentagemSuperior[20]/100);

PWM[70].i_stPara.tCyclTime:=T#10MS;
PWM[70].i_stPara.tPwmPeriod:=T#1000MS;
PWM[70](
	i_xEn:= 	xHabilitaBlocosControleSuperior,
	i_rIput:= 	rPwmEntrada[70],
	i_stPara:= 	,
	i_xErrRst:= xResetPid,
	q_xEn=> 	,
	q_xBusy=> 	,
	q_xPstv=> 	Q_xAquecimentoPwm70,
	q_xNgtv=> 	,
	q_xErr=> 	,
	q_uiErrId=> );

// Controle Resistencia 71

SR_ControleTemperatura.FbCrtlAquecimento[71](
	i_xEnable:= InterfaceHeat.P_xHabTemp71 OR xLigaDesligaSupG01,
	i_rSetPoint:= rSetPointTemperaturaSuperior[21],
	i_rProcessValue:= I_rTemperatura71,
	i_xManualMode:= ,
	i_rManualValue:= ,
	i_xAutoTune:= TEMP.xAutoTuneTemp71 OR xAutoTuneTempGeral,
	i_xHold:= ,
	i_xReset:= InterfaceHeat.xReset,
	i_stTemperatureControl:= stTemperatureControl[71],
	iq_etSelectParameterSetPID:= etSelectParameterSetPID[71],
	iq_stParameterSetsPID:= stParameterSetsPID[71],
	q_xActive=> ,
	q_xReady=> ,
	q_xError=> TEMP.xCrtlTemperatura[71],
	q_etResult=> TEMP.iCrtlTempStsTemp71,
	q_sResultMsg=> ,
	q_rAnalogOutput=> TEMP.rCrtlTempPotTemp71,
	q_xPwmOutput=> Q_xAquecimento71,
	q_xAutoTuneActive=> TEMP.xAutoTuneAtivoTemp71,
	q_etStatusAutoTune=> TEMP.iAutoTuneStsTemp71);

rPwmEntrada[71]:= TEMP.rCrtlTempPotTemp71*(rSetPorcentagemSuperior[21]/100);

PWM[71].i_stPara.tCyclTime:=T#10MS;
PWM[71].i_stPara.tPwmPeriod:=T#1000MS;
PWM[71](
	i_xEn:= 	xHabilitaBlocosControleSuperior,
	i_rIput:= 	rPwmEntrada[71],
	i_stPara:= 	,
	i_xErrRst:= xResetPid,
	q_xEn=> 	,
	q_xBusy=> 	,
	q_xPstv=> 	Q_xAquecimentoPwm71,
	q_xNgtv=> 	,
	q_xErr=> 	,
	q_uiErrId=> );

// Controle Resistencia 72

SR_ControleTemperatura.FbCrtlAquecimento[72](
	i_xEnable:= InterfaceHeat.P_xHabTemp72 OR xLigaDesligaSupG02,
	i_rSetPoint:= rSetPointTemperaturaSuperior[22],
	i_rProcessValue:= I_rTemperatura72,
	i_xManualMode:= ,
	i_rManualValue:= ,
	i_xAutoTune:= TEMP.xAutoTuneTemp72 OR xAutoTuneTempGeral,
	i_xHold:= ,
	i_xReset:= InterfaceHeat.xReset,
	i_stTemperatureControl:= stTemperatureControl[72],
	iq_etSelectParameterSetPID:= etSelectParameterSetPID[72],
	iq_stParameterSetsPID:= stParameterSetsPID[72],
	q_xActive=> ,
	q_xReady=> ,
	q_xError=> TEMP.xCrtlTemperatura[72],
	q_etResult=> TEMP.iCrtlTempStsTemp72,
	q_sResultMsg=> ,
	q_rAnalogOutput=> TEMP.rCrtlTempPotTemp72,
	q_xPwmOutput=> Q_xAquecimento72,
	q_xAutoTuneActive=> TEMP.xAutoTuneAtivoTemp72,
	q_etStatusAutoTune=> TEMP.iAutoTuneStsTemp72);

rPwmEntrada[72]:= TEMP.rCrtlTempPotTemp72*(rSetPorcentagemSuperior[22]/100);

PWM[72].i_stPara.tCyclTime:=T#10MS;
PWM[72].i_stPara.tPwmPeriod:=T#1000MS;
PWM[72](
	i_xEn:= 	xHabilitaBlocosControleSuperior,
	i_rIput:= 	rPwmEntrada[72],
	i_stPara:= 	,
	i_xErrRst:= xResetPid,
	q_xEn=> 	,
	q_xBusy=> 	,
	q_xPstv=> 	Q_xAquecimentoPwm72,
	q_xNgtv=> 	,
	q_xErr=> 	,
	q_uiErrId=> );

// Controle Resistencia 73

SR_ControleTemperatura.FbCrtlAquecimento[73](
	i_xEnable:= InterfaceHeat.P_xHabTemp73 OR xLigaDesligaSupG01,
	i_rSetPoint:= rSetPointTemperaturaSuperior[23],
	i_rProcessValue:= I_rTemperatura73,
	i_xManualMode:= ,
	i_rManualValue:= ,
	i_xAutoTune:= TEMP.xAutoTuneTemp73 OR xAutoTuneTempGeral,
	i_xHold:= ,
	i_xReset:= InterfaceHeat.xReset,
	i_stTemperatureControl:= stTemperatureControl[73],
	iq_etSelectParameterSetPID:= etSelectParameterSetPID[73],
	iq_stParameterSetsPID:= stParameterSetsPID[73],
	q_xActive=> ,
	q_xReady=> ,
	q_xError=> TEMP.xCrtlTemperatura[73],
	q_etResult=> TEMP.iCrtlTempStsTemp73,
	q_sResultMsg=> ,
	q_rAnalogOutput=> TEMP.rCrtlTempPotTemp73,
	q_xPwmOutput=> Q_xAquecimento73,
	q_xAutoTuneActive=> TEMP.xAutoTuneAtivoTemp73,
	q_etStatusAutoTune=> TEMP.iAutoTuneStsTemp73);

rPwmEntrada[73]:= TEMP.rCrtlTempPotTemp73*(rSetPorcentagemSuperior[23]/100);

PWM[73].i_stPara.tCyclTime:=T#10MS;
PWM[73].i_stPara.tPwmPeriod:=T#1000MS;
PWM[73](
	i_xEn:= 	xHabilitaBlocosControleSuperior,
	i_rIput:= 	rPwmEntrada[73],
	i_stPara:= 	,
	i_xErrRst:= xResetPid,
	q_xEn=> 	,
	q_xBusy=> 	,
	q_xPstv=> 	Q_xAquecimentoPwm73,
	q_xNgtv=> 	,
	q_xErr=> 	,
	q_uiErrId=> );

// Controle Resistencia 74

SR_ControleTemperatura.FbCrtlAquecimento[74](
	i_xEnable:= InterfaceHeat.P_xHabTemp74 OR xLigaDesligaSupG02,
	i_rSetPoint:= rSetPointTemperaturaSuperior[24],
	i_rProcessValue:= I_rTemperatura74,
	i_xManualMode:= ,
	i_rManualValue:= ,
	i_xAutoTune:= TEMP.xAutoTuneTemp74 OR xAutoTuneTempGeral,
	i_xHold:= ,
	i_xReset:= InterfaceHeat.xReset,
	i_stTemperatureControl:= stTemperatureControl[74],
	iq_etSelectParameterSetPID:= etSelectParameterSetPID[74],
	iq_stParameterSetsPID:= stParameterSetsPID[74],
	q_xActive=> ,
	q_xReady=> ,
	q_xError=> TEMP.xCrtlTemperatura[74],
	q_etResult=> TEMP.iCrtlTempStsTemp74,
	q_sResultMsg=> ,
	q_rAnalogOutput=> TEMP.rCrtlTempPotTemp74,
	q_xPwmOutput=> Q_xAquecimento74,
	q_xAutoTuneActive=> TEMP.xAutoTuneAtivoTemp74,
	q_etStatusAutoTune=> TEMP.iAutoTuneStsTemp74);

rPwmEntrada[74]:= TEMP.rCrtlTempPotTemp74*(rSetPorcentagemSuperior[24]/100);

PWM[74].i_stPara.tCyclTime:=T#10MS;
PWM[74].i_stPara.tPwmPeriod:=T#1000MS;
PWM[74](
	i_xEn:= 	xHabilitaBlocosControleSuperior,
	i_rIput:= 	rPwmEntrada[74],
	i_stPara:= 	,
	i_xErrRst:= xResetPid,
	q_xEn=> 	,
	q_xBusy=> 	,
	q_xPstv=> 	Q_xAquecimentoPwm74,
	q_xNgtv=> 	,
	q_xErr=> 	,
	q_uiErrId=> );

// Controle Resistencia 75

FbAqueceRampa[75](
	iTermopar:= TermoparLogicoSuperior[25],
	rSpTemperatura:= rSetPointTemperaturaSuperior[25],
	iTempoEstab:= iTempoEstabRampa,
	xReset:= ,
	xStartRampaCiclo=> ,
	xRampaAtiva=> xRampaAqAtiva[75],
	TemperUp=> ,
	TemperDown=> ,
	rSpTemperaturaUp=> ,
	rSetTemperaturaRampa=> rSetTemperaturaRampaAq[75] );

SR_ControleTemperatura.FbCrtlAquecimento[75](
	i_xEnable:= InterfaceHeat.P_xHabTemp75 OR xLigaDesligaSupG01,
	i_rSetPoint:= rSetPointTemperaturaSuperior[25],
	i_rProcessValue:= I_rTemperatura75,
	i_xManualMode:= ,
	i_rManualValue:= ,
	i_xAutoTune:= TEMP.xAutoTuneTemp75 OR xAutoTuneTempGeral,
	i_xHold:= ,
	i_xReset:= InterfaceHeat.xReset,
	i_stTemperatureControl:= stTemperatureControl[75],
	iq_etSelectParameterSetPID:= etSelectParameterSetPID[75],
	iq_stParameterSetsPID:= stParameterSetsPID[75],
	q_xActive=> ,
	q_xReady=> ,
	q_xError=> TEMP.xCrtlTemperatura[75],
	q_etResult=> TEMP.iCrtlTempStsTemp75,
	q_sResultMsg=> ,
	q_rAnalogOutput=> TEMP.rCrtlTempPotTemp75,
	q_xPwmOutput=> Q_xAquecimento75,
	q_xAutoTuneActive=> TEMP.xAutoTuneAtivoTemp75,
	q_etStatusAutoTune=> TEMP.iAutoTuneStsTemp75);

rPwmEntrada[75]:= TEMP.rCrtlTempPotTemp75*(rSetPorcentagemSuperior[25]/100);

PWM[75].i_stPara.tCyclTime:=T#10MS;
PWM[75].i_stPara.tPwmPeriod:=T#1000MS;
PWM[75](
	i_xEn:= 	xHabilitaBlocosControleSuperior,
	i_rIput:= 	rPwmEntrada[75],
	i_stPara:= 	,
	i_xErrRst:= xResetPid,
	q_xEn=> 	,
	q_xBusy=> 	,
	q_xPstv=> 	Q_xAquecimentoPwm75,
	q_xNgtv=> 	,
	q_xErr=> 	,
	q_uiErrId=> );

	(*IF xRampaAqAtiva[75] THEN
		xReleSsrSuperior[25]:=Q_xAquecimento75;
	ELSE
		xReleSsrSuperior[25]:=Q_xAquecimentoPwm75;
	END_IF*)

// Controle Resistencia 76

SR_ControleTemperatura.FbCrtlAquecimento[76](
	i_xEnable:= InterfaceHeat.P_xHabTemp76 OR xLigaDesligaSupG02,
	i_rSetPoint:= rSetPointTemperaturaSuperior[26],
	i_rProcessValue:= I_rTemperatura76,
	i_xManualMode:= ,
	i_rManualValue:= ,
	i_xAutoTune:= TEMP.xAutoTuneTemp76 OR xAutoTuneTempGeral,
	i_xHold:= ,
	i_xReset:= InterfaceHeat.xReset,
	i_stTemperatureControl:= stTemperatureControl[76],
	iq_etSelectParameterSetPID:= etSelectParameterSetPID[76],
	iq_stParameterSetsPID:= stParameterSetsPID[76],
	q_xActive=> ,
	q_xReady=> ,
	q_xError=> TEMP.xCrtlTemperatura[76],
	q_etResult=> TEMP.iCrtlTempStsTemp76,
	q_sResultMsg=> ,
	q_rAnalogOutput=> TEMP.rCrtlTempPotTemp76,
	q_xPwmOutput=> Q_xAquecimento76,
	q_xAutoTuneActive=> TEMP.xAutoTuneAtivoTemp76,
	q_etStatusAutoTune=> TEMP.iAutoTuneStsTemp76);

rPwmEntrada[76]:= TEMP.rCrtlTempPotTemp76*(rSetPorcentagemSuperior[26]/100);

PWM[76].i_stPara.tCyclTime:=T#10MS;
PWM[76].i_stPara.tPwmPeriod:=T#1000MS;
PWM[76](
	i_xEn:= 	xHabilitaBlocosControleSuperior,
	i_rIput:= 	rPwmEntrada[76],
	i_stPara:= 	,
	i_xErrRst:= xResetPid,
	q_xEn=> 	,
	q_xBusy=> 	,
	q_xPstv=> 	Q_xAquecimentoPwm76,
	q_xNgtv=> 	,
	q_xErr=> 	,
	q_uiErrId=> );

// Controle Resistencia 77

SR_ControleTemperatura.FbCrtlAquecimento[77](
	i_xEnable:= InterfaceHeat.P_xHabTemp77 OR xLigaDesligaSupG01,
	i_rSetPoint:= rSetPointTemperaturaSuperior[27],
	i_rProcessValue:= I_rTemperatura77,
	i_xManualMode:= ,
	i_rManualValue:= ,
	i_xAutoTune:= TEMP.xAutoTuneTemp77 OR xAutoTuneTempGeral,
	i_xHold:= ,
	i_xReset:= InterfaceHeat.xReset,
	i_stTemperatureControl:= stTemperatureControl[77],
	iq_etSelectParameterSetPID:= etSelectParameterSetPID[77],
	iq_stParameterSetsPID:= stParameterSetsPID[77],
	q_xActive=> ,
	q_xReady=> ,
	q_xError=> TEMP.xCrtlTemperatura[77],
	q_etResult=> TEMP.iCrtlTempStsTemp77,
	q_sResultMsg=> ,
	q_rAnalogOutput=> TEMP.rCrtlTempPotTemp77,
	q_xPwmOutput=> Q_xAquecimento77,
	q_xAutoTuneActive=> TEMP.xAutoTuneAtivoTemp77,
	q_etStatusAutoTune=> TEMP.iAutoTuneStsTemp77);

rPwmEntrada[77]:= TEMP.rCrtlTempPotTemp77*(rSetPorcentagemSuperior[27]/100);

PWM[77].i_stPara.tCyclTime:=T#10MS;
PWM[77].i_stPara.tPwmPeriod:=T#1000MS;
PWM[77](
	i_xEn:= 	xHabilitaBlocosControleSuperior,
	i_rIput:= 	rPwmEntrada[77],
	i_stPara:= 	,
	i_xErrRst:= xResetPid,
	q_xEn=> 	,
	q_xBusy=> 	,
	q_xPstv=> 	Q_xAquecimentoPwm77,
	q_xNgtv=> 	,
	q_xErr=> 	,
	q_uiErrId=> );

	// Controle Resistencia 78

SR_ControleTemperatura.FbCrtlAquecimento[78](
	i_xEnable:= InterfaceHeat.P_xHabTemp78 OR xLigaDesligaSupG02,
	i_rSetPoint:= rSetPointTemperaturaSuperior[28],
	i_rProcessValue:= I_rTemperatura78,
	i_xManualMode:= ,
	i_rManualValue:= ,
	i_xAutoTune:= TEMP.xAutoTuneTemp78 OR xAutoTuneTempGeral,
	i_xHold:= ,
	i_xReset:= InterfaceHeat.xReset,
	i_stTemperatureControl:= stTemperatureControl[78],
	iq_etSelectParameterSetPID:= etSelectParameterSetPID[78],
	iq_stParameterSetsPID:= stParameterSetsPID[78],
	q_xActive=> ,
	q_xReady=> ,
	q_xError=> TEMP.xCrtlTemperatura[78],
	q_etResult=> TEMP.iCrtlTempStsTemp78,
	q_sResultMsg=> ,
	q_rAnalogOutput=> TEMP.rCrtlTempPotTemp78,
	q_xPwmOutput=> Q_xAquecimento78,
	q_xAutoTuneActive=> TEMP.xAutoTuneAtivoTemp78,
	q_etStatusAutoTune=> TEMP.iAutoTuneStsTemp78);

	rPwmEntrada[78]:= TEMP.rCrtlTempPotTemp78*(rSetPorcentagemSuperior[28]/100);

PWM[78].i_stPara.tCyclTime:=T#10MS;
PWM[78].i_stPara.tPwmPeriod:=T#1000MS;
PWM[78](
	i_xEn:= 	xHabilitaBlocosControleSuperior,
	i_rIput:= 	rPwmEntrada[78],
	i_stPara:= 	,
	i_xErrRst:= xResetPid,
	q_xEn=> 	,
	q_xBusy=> 	,
	q_xPstv=> 	Q_xAquecimentoPwm78,
	q_xNgtv=> 	,
	q_xErr=> 	,
	q_uiErrId=> );

// Controle Resistencia 79

SR_ControleTemperatura.FbCrtlAquecimento[79](
	i_xEnable:= InterfaceHeat.P_xHabTemp79 OR xLigaDesligaSupG01,
	i_rSetPoint:= rSetPointTemperaturaSuperior[29],
	i_rProcessValue:= I_rTemperatura79,
	i_xManualMode:= ,
	i_rManualValue:= ,
	i_xAutoTune:= TEMP.xAutoTuneTemp79 OR xAutoTuneTempGeral,
	i_xHold:= ,
	i_xReset:= InterfaceHeat.xReset,
	i_stTemperatureControl:= stTemperatureControl[79],
	iq_etSelectParameterSetPID:= etSelectParameterSetPID[79],
	iq_stParameterSetsPID:= stParameterSetsPID[79],
	q_xActive=> ,
	q_xReady=> ,
	q_xError=> TEMP.xCrtlTemperatura[79],
	q_etResult=> TEMP.iCrtlTempStsTemp79,
	q_sResultMsg=> ,
	q_rAnalogOutput=> TEMP.rCrtlTempPotTemp79,
	q_xPwmOutput=> Q_xAquecimento79,
	q_xAutoTuneActive=> TEMP.xAutoTuneAtivoTemp79,
	q_etStatusAutoTune=> TEMP.iAutoTuneStsTemp79);

	rPwmEntrada[79]:= TEMP.rCrtlTempPotTemp79*(rSetPorcentagemSuperior[29]/100);

PWM[79].i_stPara.tCyclTime:=T#10MS;
PWM[79].i_stPara.tPwmPeriod:=T#1000MS;
PWM[79](
	i_xEn:= 	xHabilitaBlocosControleSuperior,
	i_rIput:= 	rPwmEntrada[79],
	i_stPara:= 	,
	i_xErrRst:= xResetPid,
	q_xEn=> 	,
	q_xBusy=> 	,
	q_xPstv=> 	Q_xAquecimentoPwm79,
	q_xNgtv=> 	,
	q_xErr=> 	,
	q_uiErrId=> );

// Controle Resistencia 80

SR_ControleTemperatura.FbCrtlAquecimento[80](
	i_xEnable:= InterfaceHeat.P_xHabTemp80 OR xLigaDesligaSupG02,
	i_rSetPoint:= rSetPointTemperaturaSuperior[30],
	i_rProcessValue:= I_rTemperatura80,
	i_xManualMode:= ,
	i_rManualValue:= ,
	i_xAutoTune:= TEMP.xAutoTuneTemp80 OR xAutoTuneTempGeral,
	i_xHold:= ,
	i_xReset:= InterfaceHeat.xReset,
	i_stTemperatureControl:= stTemperatureControl[80],
	iq_etSelectParameterSetPID:= etSelectParameterSetPID[80],
	iq_stParameterSetsPID:= stParameterSetsPID[80],
	q_xActive=> ,
	q_xReady=> ,
	q_xError=> TEMP.xCrtlTemperatura[80],
	q_etResult=> TEMP.iCrtlTempStsTemp80,
	q_sResultMsg=> ,
	q_rAnalogOutput=> TEMP.rCrtlTempPotTemp80,
	q_xPwmOutput=> Q_xAquecimento80,
	q_xAutoTuneActive=> TEMP.xAutoTuneAtivoTemp80,
	q_etStatusAutoTune=> TEMP.iAutoTuneStsTemp80);

rPwmEntrada[80]:= TEMP.rCrtlTempPotTemp80*(rSetPorcentagemSuperior[30]/100);

PWM[80].i_stPara.tCyclTime:=T#10MS;
PWM[80].i_stPara.tPwmPeriod:=T#1000MS;
PWM[80](
	i_xEn:= 	xHabilitaBlocosControleSuperior,
	i_rIput:= 	rPwmEntrada[80],
	i_stPara:= 	,
	i_xErrRst:= xResetPid,
	q_xEn=> 	,
	q_xBusy=> 	,
	q_xPstv=> 	Q_xAquecimentoPwm80,
	q_xNgtv=> 	,
	q_xErr=> 	,
	q_uiErrId=> );

// Controle Resistencia 81

SR_ControleTemperatura.FbCrtlAquecimento[81](
	i_xEnable:= InterfaceHeat.P_xHabTemp81 OR xLigaDesligaSupG02,
	i_rSetPoint:= rSetPointTemperaturaSuperior[31],
	i_rProcessValue:= I_rTemperatura81,
	i_xManualMode:= ,
	i_rManualValue:= ,
	i_xAutoTune:= TEMP.xAutoTuneTemp81 OR xAutoTuneTempGeral,
	i_xHold:= ,
	i_xReset:= InterfaceHeat.xReset,
	i_stTemperatureControl:= stTemperatureControl[81],
	iq_etSelectParameterSetPID:= etSelectParameterSetPID[81],
	iq_stParameterSetsPID:= stParameterSetsPID[81],
	q_xActive=> ,
	q_xReady=> ,
	q_xError=> TEMP.xCrtlTemperatura[81],
	q_etResult=> TEMP.iCrtlTempStsTemp81,
	q_sResultMsg=> ,
	q_rAnalogOutput=> TEMP.rCrtlTempPotTemp81,
	q_xPwmOutput=> Q_xAquecimento81,
	q_xAutoTuneActive=> TEMP.xAutoTuneAtivoTemp81,
	q_etStatusAutoTune=> TEMP.iAutoTuneStsTemp81);

rPwmEntrada[81]:= TEMP.rCrtlTempPotTemp81*(rSetPorcentagemSuperior[31]/100);

PWM[81].i_stPara.tCyclTime:=T#10MS;
PWM[81].i_stPara.tPwmPeriod:=T#1000MS;
PWM[81](
	i_xEn:= 	xHabilitaBlocosControleSuperior,
	i_rIput:= 	rPwmEntrada[81],
	i_stPara:= 	,
	i_xErrRst:= xResetPid,
	q_xEn=> 	,
	q_xBusy=> 	,
	q_xPstv=> 	Q_xAquecimentoPwm81,
	q_xNgtv=> 	,
	q_xErr=> 	,
	q_uiErrId=> );

// Controle Resistencia 82

SR_ControleTemperatura.FbCrtlAquecimento[82](
	i_xEnable:= InterfaceHeat.P_xHabTemp82 OR xLigaDesligaSupG01,
	i_rSetPoint:= rSetPointTemperaturaSuperior[32],
	i_rProcessValue:= I_rTemperatura82,
	i_xManualMode:= ,
	i_rManualValue:= ,
	i_xAutoTune:= TEMP.xAutoTuneTemp82 OR xAutoTuneTempGeral,
	i_xHold:= ,
	i_xReset:= InterfaceHeat.xReset,
	i_stTemperatureControl:= stTemperatureControl[82],
	iq_etSelectParameterSetPID:= etSelectParameterSetPID[82],
	iq_stParameterSetsPID:= stParameterSetsPID[82],
	q_xActive=> ,
	q_xReady=> ,
	q_xError=> TEMP.xCrtlTemperatura[82],
	q_etResult=> TEMP.iCrtlTempStsTemp82,
	q_sResultMsg=> ,
	q_rAnalogOutput=> TEMP.rCrtlTempPotTemp82,
	q_xPwmOutput=> Q_xAquecimento82,
	q_xAutoTuneActive=> TEMP.xAutoTuneAtivoTemp82,
	q_etStatusAutoTune=> TEMP.iAutoTuneStsTemp82);

rPwmEntrada[82]:= TEMP.rCrtlTempPotTemp82*(rSetPorcentagemSuperior[32]/100);

PWM[82].i_stPara.tCyclTime:=T#10MS;
PWM[82].i_stPara.tPwmPeriod:=T#1000MS;
PWM[82](
	i_xEn:= 	xHabilitaBlocosControleSuperior,
	i_rIput:= 	rPwmEntrada[82],
	i_stPara:= 	,
	i_xErrRst:= xResetPid,
	q_xEn=> 	,
	q_xBusy=> 	,
	q_xPstv=> 	Q_xAquecimentoPwm82,
	q_xNgtv=> 	,
	q_xErr=> 	,
	q_uiErrId=> );

// Controle Resistencia 83

SR_ControleTemperatura.FbCrtlAquecimento[83](
	i_xEnable:= InterfaceHeat.P_xHabTemp83 OR xLigaDesligaSupG02,
	i_rSetPoint:= rSetPointTemperaturaSuperior[33],
	i_rProcessValue:= I_rTemperatura83,
	i_xManualMode:= ,
	i_rManualValue:= ,
	i_xAutoTune:= TEMP.xAutoTuneTemp83 OR xAutoTuneTempGeral,
	i_xHold:= ,
	i_xReset:= InterfaceHeat.xReset,
	i_stTemperatureControl:= stTemperatureControl[83],
	iq_etSelectParameterSetPID:= etSelectParameterSetPID[83],
	iq_stParameterSetsPID:= stParameterSetsPID[83],
	q_xActive=> ,
	q_xReady=> ,
	q_xError=> TEMP.xCrtlTemperatura[83],
	q_etResult=> TEMP.iCrtlTempStsTemp83,
	q_sResultMsg=> ,
	q_rAnalogOutput=> TEMP.rCrtlTempPotTemp83,
	q_xPwmOutput=> Q_xAquecimento83,
	q_xAutoTuneActive=> TEMP.xAutoTuneAtivoTemp83,
	q_etStatusAutoTune=> TEMP.iAutoTuneStsTemp83);

rPwmEntrada[83]:= TEMP.rCrtlTempPotTemp83*(rSetPorcentagemSuperior[33]/100);

PWM[83].i_stPara.tCyclTime:=T#10MS;
PWM[83].i_stPara.tPwmPeriod:=T#1000MS;
PWM[83](
	i_xEn:= 	xHabilitaBlocosControleSuperior,
	i_rIput:= 	rPwmEntrada[83],
	i_stPara:= 	,
	i_xErrRst:= xResetPid,
	q_xEn=> 	,
	q_xBusy=> 	,
	q_xPstv=> 	Q_xAquecimentoPwm83,
	q_xNgtv=> 	,
	q_xErr=> 	,
	q_uiErrId=> );

// Controle Resistencia 84

SR_ControleTemperatura.FbCrtlAquecimento[84](
	i_xEnable:= InterfaceHeat.P_xHabTemp84 OR xLigaDesligaSupG01,
	i_rSetPoint:= rSetPointTemperaturaSuperior[34],
	i_rProcessValue:= I_rTemperatura84,
	i_xManualMode:= ,
	i_rManualValue:= ,
	i_xAutoTune:= TEMP.xAutoTuneTemp84 OR xAutoTuneTempGeral,
	i_xHold:= ,
	i_xReset:= InterfaceHeat.xReset,
	i_stTemperatureControl:= stTemperatureControl[84],
	iq_etSelectParameterSetPID:= etSelectParameterSetPID[84],
	iq_stParameterSetsPID:= stParameterSetsPID[84],
	q_xActive=> ,
	q_xReady=> ,
	q_xError=> TEMP.xCrtlTemperatura[84],
	q_etResult=> TEMP.iCrtlTempStsTemp84,
	q_sResultMsg=> ,
	q_rAnalogOutput=> TEMP.rCrtlTempPotTemp84,
	q_xPwmOutput=> Q_xAquecimento84,
	q_xAutoTuneActive=> TEMP.xAutoTuneAtivoTemp84,
	q_etStatusAutoTune=> TEMP.iAutoTuneStsTemp84);

rPwmEntrada[84]:= TEMP.rCrtlTempPotTemp84*(rSetPorcentagemSuperior[34]/100);

PWM[84].i_stPara.tCyclTime:=T#10MS;
PWM[84].i_stPara.tPwmPeriod:=T#1000MS;
PWM[84](
	i_xEn:= 	xHabilitaBlocosControleSuperior,
	i_rIput:= 	rPwmEntrada[84],
	i_stPara:= 	,
	i_xErrRst:= xResetPid,
	q_xEn=> 	,
	q_xBusy=> 	,
	q_xPstv=> 	Q_xAquecimentoPwm84,
	q_xNgtv=> 	,
	q_xErr=> 	,
	q_uiErrId=> );

// Controle Resistencia 85

SR_ControleTemperatura.FbCrtlAquecimento[85](
	i_xEnable:= InterfaceHeat.P_xHabTemp85 OR xLigaDesligaSupG02,
	i_rSetPoint:= rSetPointTemperaturaSuperior[35],
	i_rProcessValue:= I_rTemperatura85,
	i_xManualMode:= ,
	i_rManualValue:= ,
	i_xAutoTune:= TEMP.xAutoTuneTemp85 OR xAutoTuneTempGeral,
	i_xHold:= ,
	i_xReset:= InterfaceHeat.xReset,
	i_stTemperatureControl:= stTemperatureControl[85],
	iq_etSelectParameterSetPID:= etSelectParameterSetPID[85],
	iq_stParameterSetsPID:= stParameterSetsPID[85],
	q_xActive=> ,
	q_xReady=> ,
	q_xError=> TEMP.xCrtlTemperatura[85],
	q_etResult=> TEMP.iCrtlTempStsTemp85,
	q_sResultMsg=> ,
	q_rAnalogOutput=> TEMP.rCrtlTempPotTemp85,
	q_xPwmOutput=> Q_xAquecimento85,
	q_xAutoTuneActive=> TEMP.xAutoTuneAtivoTemp85,
	q_etStatusAutoTune=> TEMP.iAutoTuneStsTemp85);

rPwmEntrada[85]:= TEMP.rCrtlTempPotTemp85*(rSetPorcentagemSuperior[35]/100);

PWM[85].i_stPara.tCyclTime:=T#10MS;
PWM[85].i_stPara.tPwmPeriod:=T#1000MS;
PWM[85](
	i_xEn:= 	xHabilitaBlocosControleSuperior,
	i_rIput:= 	rPwmEntrada[85],
	i_stPara:= 	,
	i_xErrRst:= xResetPid,
	q_xEn=> 	,
	q_xBusy=> 	,
	q_xPstv=> 	Q_xAquecimentoPwm85,
	q_xNgtv=> 	,
	q_xErr=> 	,
	q_uiErrId=> );

// Controle Resistencia 86

SR_ControleTemperatura.FbCrtlAquecimento[86](
	i_xEnable:= InterfaceHeat.P_xHabTemp86 OR xLigaDesligaSupG01,
	i_rSetPoint:= rSetPointTemperaturaSuperior[36],
	i_rProcessValue:= I_rTemperatura86,
	i_xManualMode:= ,
	i_rManualValue:= ,
	i_xAutoTune:= TEMP.xAutoTuneTemp86 OR xAutoTuneTempGeral,
	i_xHold:= ,
	i_xReset:= InterfaceHeat.xReset,
	i_stTemperatureControl:= stTemperatureControl[86],
	iq_etSelectParameterSetPID:= etSelectParameterSetPID[86],
	iq_stParameterSetsPID:= stParameterSetsPID[86],
	q_xActive=> ,
	q_xReady=> ,
	q_xError=> TEMP.xCrtlTemperatura[86],
	q_etResult=> TEMP.iCrtlTempStsTemp86,
	q_sResultMsg=> ,
	q_rAnalogOutput=> TEMP.rCrtlTempPotTemp86,
	q_xPwmOutput=> Q_xAquecimento86,
	q_xAutoTuneActive=> TEMP.xAutoTuneAtivoTemp86,
	q_etStatusAutoTune=> TEMP.iAutoTuneStsTemp86);

rPwmEntrada[86]:= TEMP.rCrtlTempPotTemp86*(rSetPorcentagemSuperior[36]/100);

PWM[86].i_stPara.tCyclTime:=T#10MS;
PWM[86].i_stPara.tPwmPeriod:=T#1000MS;
PWM[86](
	i_xEn:= 	xHabilitaBlocosControleSuperior,
	i_rIput:= 	rPwmEntrada[86],
	i_stPara:= 	,
	i_xErrRst:= xResetPid,
	q_xEn=> 	,
	q_xBusy=> 	,
	q_xPstv=> 	Q_xAquecimentoPwm86,
	q_xNgtv=> 	,
	q_xErr=> 	,
	q_uiErrId=> );

// Controle Resistencia 87

SR_ControleTemperatura.FbCrtlAquecimento[87](
	i_xEnable:= InterfaceHeat.P_xHabTemp87 OR xLigaDesligaSupG02,
	i_rSetPoint:= rSetPointTemperaturaSuperior[37],
	i_rProcessValue:= I_rTemperatura87,
	i_xManualMode:= ,
	i_rManualValue:= ,
	i_xAutoTune:= TEMP.xAutoTuneTemp87 OR xAutoTuneTempGeral,
	i_xHold:= ,
	i_xReset:= InterfaceHeat.xReset,
	i_stTemperatureControl:= stTemperatureControl[87],
	iq_etSelectParameterSetPID:= etSelectParameterSetPID[87],
	iq_stParameterSetsPID:= stParameterSetsPID[87],
	q_xActive=> ,
	q_xReady=> ,
	q_xError=> TEMP.xCrtlTemperatura[87],
	q_etResult=> TEMP.iCrtlTempStsTemp87,
	q_sResultMsg=> ,
	q_rAnalogOutput=> TEMP.rCrtlTempPotTemp87,
	q_xPwmOutput=> Q_xAquecimento87,
	q_xAutoTuneActive=> TEMP.xAutoTuneAtivoTemp87,
	q_etStatusAutoTune=> TEMP.iAutoTuneStsTemp87);

	rPwmEntrada[87]:= TEMP.rCrtlTempPotTemp87*(rSetPorcentagemSuperior[37]/100);

PWM[87].i_stPara.tCyclTime:=T#10MS;
PWM[87].i_stPara.tPwmPeriod:=T#1000MS;
PWM[87](
	i_xEn:= 	xHabilitaBlocosControleSuperior,
	i_rIput:= 	rPwmEntrada[87],
	i_stPara:= 	,
	i_xErrRst:= xResetPid,
	q_xEn=> 	,
	q_xBusy=> 	,
	q_xPstv=> 	Q_xAquecimentoPwm87,
	q_xNgtv=> 	,
	q_xErr=> 	,
	q_uiErrId=> );

// Controle Resistencia 88

SR_ControleTemperatura.FbCrtlAquecimento[88](
	i_xEnable:= InterfaceHeat.P_xHabTemp88 OR xLigaDesligaSupG01,
	i_rSetPoint:= rSetPointTemperaturaSuperior[38],
	i_rProcessValue:= I_rTemperatura88,
	i_xManualMode:= ,
	i_rManualValue:= ,
	i_xAutoTune:= TEMP.xAutoTuneTemp88 OR xAutoTuneTempGeral,
	i_xHold:= ,
	i_xReset:= InterfaceHeat.xReset,
	i_stTemperatureControl:= stTemperatureControl[88],
	iq_etSelectParameterSetPID:= etSelectParameterSetPID[88],
	iq_stParameterSetsPID:= stParameterSetsPID[88],
	q_xActive=> ,
	q_xReady=> ,
	q_xError=> TEMP.xCrtlTemperatura[88],
	q_etResult=> TEMP.iCrtlTempStsTemp88,
	q_sResultMsg=> ,
	q_rAnalogOutput=> TEMP.rCrtlTempPotTemp88,
	q_xPwmOutput=> Q_xAquecimento88,
	q_xAutoTuneActive=> TEMP.xAutoTuneAtivoTemp88,
	q_etStatusAutoTune=> TEMP.iAutoTuneStsTemp88);

rPwmEntrada[88]:= TEMP.rCrtlTempPotTemp88*(rSetPorcentagemSuperior[38]/100);

PWM[88].i_stPara.tCyclTime:=T#10MS;
PWM[88].i_stPara.tPwmPeriod:=T#1000MS;
PWM[88](
	i_xEn:= 	xHabilitaBlocosControleSuperior,
	i_rIput:= 	rPwmEntrada[88],
	i_stPara:= 	,
	i_xErrRst:= xResetPid,
	q_xEn=> 	,
	q_xBusy=> 	,
	q_xPstv=> 	Q_xAquecimentoPwm88,
	q_xNgtv=> 	,
	q_xErr=> 	,
	q_uiErrId=> );

	// Controle Resistencia 89

SR_ControleTemperatura.FbCrtlAquecimento[89](
	i_xEnable:= InterfaceHeat.P_xHabTemp89 OR xLigaDesligaSupG02,
	i_rSetPoint:= rSetPointTemperaturaSuperior[39],
	i_rProcessValue:= I_rTemperatura89,
	i_xManualMode:= ,
	i_rManualValue:= ,
	i_xAutoTune:= TEMP.xAutoTuneTemp89 OR xAutoTuneTempGeral,
	i_xHold:= ,
	i_xReset:= InterfaceHeat.xReset,
	i_stTemperatureControl:= stTemperatureControl[89],
	iq_etSelectParameterSetPID:= etSelectParameterSetPID[89],
	iq_stParameterSetsPID:= stParameterSetsPID[89],
	q_xActive=> ,
	q_xReady=> ,
	q_xError=> TEMP.xCrtlTemperatura[89],
	q_etResult=> TEMP.iCrtlTempStsTemp89,
	q_sResultMsg=> ,
	q_rAnalogOutput=> TEMP.rCrtlTempPotTemp89,
	q_xPwmOutput=> Q_xAquecimento89,
	q_xAutoTuneActive=> TEMP.xAutoTuneAtivoTemp89,
	q_etStatusAutoTune=> TEMP.iAutoTuneStsTemp89);

rPwmEntrada[89]:= TEMP.rCrtlTempPotTemp89*(rSetPorcentagemSuperior[39]/100);

PWM[89].i_stPara.tCyclTime:=T#10MS;
PWM[89].i_stPara.tPwmPeriod:=T#1000MS;
PWM[89](
	i_xEn:= 	xHabilitaBlocosControleSuperior,
	i_rIput:= 	rPwmEntrada[89],
	i_stPara:= 	,
	i_xErrRst:= xResetPid,
	q_xEn=> 	,
	q_xBusy=> 	,
	q_xPstv=> 	Q_xAquecimentoPwm89,
	q_xNgtv=> 	,
	q_xErr=> 	,
	q_uiErrId=> );

	// Controle Resistencia 90

SR_ControleTemperatura.FbCrtlAquecimento[90](
	i_xEnable:= InterfaceHeat.P_xHabTemp90 OR xLigaDesligaSupG01,
	i_rSetPoint:= rSetPointTemperaturaSuperior[40],
	i_rProcessValue:= I_rTemperatura90,
	i_xManualMode:= ,
	i_rManualValue:= ,
	i_xAutoTune:= TEMP.xAutoTuneTemp90 OR xAutoTuneTempGeral,
	i_xHold:= ,
	i_xReset:= InterfaceHeat.xReset,
	i_stTemperatureControl:= stTemperatureControl[90],
	iq_etSelectParameterSetPID:= etSelectParameterSetPID[90],
	iq_stParameterSetsPID:= stParameterSetsPID[90],
	q_xActive=> ,
	q_xReady=> ,
	q_xError=> TEMP.xCrtlTemperatura[90],
	q_etResult=> TEMP.iCrtlTempStsTemp90,
	q_sResultMsg=> ,
	q_rAnalogOutput=> TEMP.rCrtlTempPotTemp90,
	q_xPwmOutput=> Q_xAquecimento90,
	q_xAutoTuneActive=> TEMP.xAutoTuneAtivoTemp90,
	q_etStatusAutoTune=> TEMP.iAutoTuneStsTemp90);

rPwmEntrada[90]:= TEMP.rCrtlTempPotTemp90*(rSetPorcentagemSuperior[40]/100);

PWM[90].i_stPara.tCyclTime:=T#10MS;
PWM[90].i_stPara.tPwmPeriod:=T#1000MS;
PWM[90](
	i_xEn:= 	xHabilitaBlocosControleSuperior,
	i_rIput:= 	rPwmEntrada[90],
	i_stPara:= 	,
	i_xErrRst:= xResetPid,
	q_xEn=> 	,
	q_xBusy=> 	,
	q_xPstv=> 	Q_xAquecimentoPwm90,
	q_xNgtv=> 	,
	q_xErr=> 	,
	q_uiErrId=> );

// Controle Resistencia 91

SR_ControleTemperatura.FbCrtlAquecimento[91](
	i_xEnable:= InterfaceHeat.P_xHabTemp91 OR xLigaDesligaSupG01,
	i_rSetPoint:= rSetPointTemperaturaSuperior[41],
	i_rProcessValue:= I_rTemperatura91,
	i_xManualMode:= ,
	i_rManualValue:= ,
	i_xAutoTune:= TEMP.xAutoTuneTemp91 OR xAutoTuneTempGeral,
	i_xHold:= ,
	i_xReset:= InterfaceHeat.xReset,
	i_stTemperatureControl:= stTemperatureControl[91],
	iq_etSelectParameterSetPID:= etSelectParameterSetPID[91],
	iq_stParameterSetsPID:= stParameterSetsPID[91],
	q_xActive=> ,
	q_xReady=> ,
	q_xError=> TEMP.xCrtlTemperatura[91],
	q_etResult=> TEMP.iCrtlTempStsTemp91,
	q_sResultMsg=> ,
	q_rAnalogOutput=> TEMP.rCrtlTempPotTemp91,
	q_xPwmOutput=> Q_xAquecimento91,
	q_xAutoTuneActive=> TEMP.xAutoTuneAtivoTemp91,
	q_etStatusAutoTune=> TEMP.iAutoTuneStsTemp91);

rPwmEntrada[91]:= TEMP.rCrtlTempPotTemp91*(rSetPorcentagemSuperior[41]/100);

PWM[91].i_stPara.tCyclTime:=T#10MS;
PWM[91].i_stPara.tPwmPeriod:=T#1000MS;
PWM[91](
	i_xEn:= 	xHabilitaBlocosControleSuperior,
	i_rIput:= 	rPwmEntrada[91],
	i_stPara:= 	,
	i_xErrRst:= xResetPid,
	q_xEn=> 	,
	q_xBusy=> 	,
	q_xPstv=> 	Q_xAquecimentoPwm91,
	q_xNgtv=> 	,
	q_xErr=> 	,
	q_uiErrId=> );

// Controle Resistencia 92

SR_ControleTemperatura.FbCrtlAquecimento[92](
	i_xEnable:= InterfaceHeat.P_xHabTemp92 OR xLigaDesligaSupG02,
	i_rSetPoint:= rSetPointTemperaturaSuperior[42],
	i_rProcessValue:= I_rTemperatura92,
	i_xManualMode:= ,
	i_rManualValue:= ,
	i_xAutoTune:= TEMP.xAutoTuneTemp92 OR xAutoTuneTempGeral,
	i_xHold:= ,
	i_xReset:= InterfaceHeat.xReset,
	i_stTemperatureControl:= stTemperatureControl[92],
	iq_etSelectParameterSetPID:= etSelectParameterSetPID[92],
	iq_stParameterSetsPID:= stParameterSetsPID[92],
	q_xActive=> ,
	q_xReady=> ,
	q_xError=> TEMP.xCrtlTemperatura[92],
	q_etResult=> TEMP.iCrtlTempStsTemp92,
	q_sResultMsg=> ,
	q_rAnalogOutput=> TEMP.rCrtlTempPotTemp92,
	q_xPwmOutput=> Q_xAquecimento92,
	q_xAutoTuneActive=> TEMP.xAutoTuneAtivoTemp92,
	q_etStatusAutoTune=> TEMP.iAutoTuneStsTemp92);

rPwmEntrada[92]:= TEMP.rCrtlTempPotTemp92*(rSetPorcentagemSuperior[42]/100);

PWM[92].i_stPara.tCyclTime:=T#10MS;
PWM[92].i_stPara.tPwmPeriod:=T#1000MS;
PWM[92](
	i_xEn:= 	xHabilitaBlocosControleSuperior,
	i_rIput:= 	rPwmEntrada[92],
	i_stPara:= 	,
	i_xErrRst:= xResetPid,
	q_xEn=> 	,
	q_xBusy=> 	,
	q_xPstv=> 	Q_xAquecimentoPwm92,
	q_xNgtv=> 	,
	q_xErr=> 	,
	q_uiErrId=> );

// Controle Resistencia 93

SR_ControleTemperatura.FbCrtlAquecimento[93](
	i_xEnable:= InterfaceHeat.P_xHabTemp93 OR xLigaDesligaSupG01,
	i_rSetPoint:= rSetPointTemperaturaSuperior[43],
	i_rProcessValue:= I_rTemperatura93,
	i_xManualMode:= ,
	i_rManualValue:= ,
	i_xAutoTune:= TEMP.xAutoTuneTemp93 OR xAutoTuneTempGeral,
	i_xHold:= ,
	i_xReset:= InterfaceHeat.xReset,
	i_stTemperatureControl:= stTemperatureControl[93],
	iq_etSelectParameterSetPID:= etSelectParameterSetPID[93],
	iq_stParameterSetsPID:= stParameterSetsPID[93],
	q_xActive=> ,
	q_xReady=> ,
	q_xError=> TEMP.xCrtlTemperatura[93],
	q_etResult=> TEMP.iCrtlTempStsTemp93,
	q_sResultMsg=> ,
	q_rAnalogOutput=> TEMP.rCrtlTempPotTemp93,
	q_xPwmOutput=> Q_xAquecimento93,
	q_xAutoTuneActive=> TEMP.xAutoTuneAtivoTemp93,
	q_etStatusAutoTune=> TEMP.iAutoTuneStsTemp93);

rPwmEntrada[93]:= TEMP.rCrtlTempPotTemp93*(rSetPorcentagemSuperior[43]/100);

PWM[93].i_stPara.tCyclTime:=T#10MS;
PWM[93].i_stPara.tPwmPeriod:=T#1000MS;
PWM[93](
	i_xEn:= 	xHabilitaBlocosControleSuperior,
	i_rIput:= 	rPwmEntrada[93],
	i_stPara:= 	,
	i_xErrRst:= xResetPid,
	q_xEn=> 	,
	q_xBusy=> 	,
	q_xPstv=> 	Q_xAquecimentoPwm93,
	q_xNgtv=> 	,
	q_xErr=> 	,
	q_uiErrId=> );

// Controle Resistencia 94

SR_ControleTemperatura.FbCrtlAquecimento[94](
	i_xEnable:= InterfaceHeat.P_xHabTemp94 OR xLigaDesligaSupG02,
	i_rSetPoint:= rSetPointTemperaturaSuperior[44],
	i_rProcessValue:= I_rTemperatura94,
	i_xManualMode:= ,
	i_rManualValue:= ,
	i_xAutoTune:= TEMP.xAutoTuneTemp94 OR xAutoTuneTempGeral,
	i_xHold:= ,
	i_xReset:= InterfaceHeat.xReset,
	i_stTemperatureControl:= stTemperatureControl[94],
	iq_etSelectParameterSetPID:= etSelectParameterSetPID[94],
	iq_stParameterSetsPID:= stParameterSetsPID[94],
	q_xActive=> ,
	q_xReady=> ,
	q_xError=> TEMP.xCrtlTemperatura[94],
	q_etResult=> TEMP.iCrtlTempStsTemp94,
	q_sResultMsg=> ,
	q_rAnalogOutput=> TEMP.rCrtlTempPotTemp94,
	q_xPwmOutput=> Q_xAquecimento94,
	q_xAutoTuneActive=> TEMP.xAutoTuneAtivoTemp94,
	q_etStatusAutoTune=> TEMP.iAutoTuneStsTemp94);

rPwmEntrada[94]:= TEMP.rCrtlTempPotTemp94*(rSetPorcentagemSuperior[44]/100);

PWM[94].i_stPara.tCyclTime:=T#10MS;
PWM[94].i_stPara.tPwmPeriod:=T#1000MS;
PWM[94](
	i_xEn:= 	xHabilitaBlocosControleSuperior,
	i_rIput:= 	rPwmEntrada[94],
	i_stPara:= 	,
	i_xErrRst:= xResetPid,
	q_xEn=> 	,
	q_xBusy=> 	,
	q_xPstv=> 	Q_xAquecimentoPwm94,
	q_xNgtv=> 	,
	q_xErr=> 	,
	q_uiErrId=> );

// Controle Resistencia 95

SR_ControleTemperatura.FbCrtlAquecimento[95](
	i_xEnable:= InterfaceHeat.P_xHabTemp95 OR xLigaDesligaSupG01,
	i_rSetPoint:= rSetPointTemperaturaSuperior[45],
	i_rProcessValue:= I_rTemperatura95,
	i_xManualMode:= ,
	i_rManualValue:= ,
	i_xAutoTune:= TEMP.xAutoTuneTemp95 OR xAutoTuneTempGeral,
	i_xHold:= ,
	i_xReset:= InterfaceHeat.xReset,
	i_stTemperatureControl:= stTemperatureControl[95],
	iq_etSelectParameterSetPID:= etSelectParameterSetPID[95],
	iq_stParameterSetsPID:= stParameterSetsPID[95],
	q_xActive=> ,
	q_xReady=> ,
	q_xError=> TEMP.xCrtlTemperatura[95],
	q_etResult=> TEMP.iCrtlTempStsTemp95,
	q_sResultMsg=> ,
	q_rAnalogOutput=> TEMP.rCrtlTempPotTemp95,
	q_xPwmOutput=> Q_xAquecimento95,
	q_xAutoTuneActive=> TEMP.xAutoTuneAtivoTemp95,
	q_etStatusAutoTune=> TEMP.iAutoTuneStsTemp95);

rPwmEntrada[95]:= TEMP.rCrtlTempPotTemp95*(rSetPorcentagemSuperior[45]/100);

PWM[95].i_stPara.tCyclTime:=T#10MS;
PWM[95].i_stPara.tPwmPeriod:=T#1000MS;
PWM[95](
	i_xEn:= 	xHabilitaBlocosControleSuperior,
	i_rIput:= 	rPwmEntrada[95],
	i_stPara:= 	,
	i_xErrRst:= xResetPid,
	q_xEn=> 	,
	q_xBusy=> 	,
	q_xPstv=> 	Q_xAquecimentoPwm95,
	q_xNgtv=> 	,
	q_xErr=> 	,
	q_uiErrId=> );

// Controle Resistencia 96

SR_ControleTemperatura.FbCrtlAquecimento[96](
	i_xEnable:= InterfaceHeat.P_xHabTemp96 OR xLigaDesligaSupG02,
	i_rSetPoint:= rSetPointTemperaturaSuperior[46],
	i_rProcessValue:= I_rTemperatura96,
	i_xManualMode:= ,
	i_rManualValue:= ,
	i_xAutoTune:= TEMP.xAutoTuneTemp96 OR xAutoTuneTempGeral,
	i_xHold:= ,
	i_xReset:= InterfaceHeat.xReset,
	i_stTemperatureControl:= stTemperatureControl[96],
	iq_etSelectParameterSetPID:= etSelectParameterSetPID[96],
	iq_stParameterSetsPID:= stParameterSetsPID[96],
	q_xActive=> ,
	q_xReady=> ,
	q_xError=> TEMP.xCrtlTemperatura[96],
	q_etResult=> TEMP.iCrtlTempStsTemp96,
	q_sResultMsg=> ,
	q_rAnalogOutput=> TEMP.rCrtlTempPotTemp96,
	q_xPwmOutput=> Q_xAquecimento96,
	q_xAutoTuneActive=> TEMP.xAutoTuneAtivoTemp96,
	q_etStatusAutoTune=> TEMP.iAutoTuneStsTemp96);

rPwmEntrada[96]:= TEMP.rCrtlTempPotTemp96*(rSetPorcentagemSuperior[46]/100);

PWM[96].i_stPara.tCyclTime:=T#10MS;
PWM[96].i_stPara.tPwmPeriod:=T#1000MS;
PWM[96](
	i_xEn:= 	xHabilitaBlocosControleSuperior,
	i_rIput:= 	rPwmEntrada[96],
	i_stPara:= 	,
	i_xErrRst:= xResetPid,
	q_xEn=> 	,
	q_xBusy=> 	,
	q_xPstv=> 	Q_xAquecimentoPwm96,
	q_xNgtv=> 	,
	q_xErr=> 	,
	q_uiErrId=> );

// Controle Resistencia 97

SR_ControleTemperatura.FbCrtlAquecimento[97](
	i_xEnable:= InterfaceHeat.P_xHabTemp97 OR xLigaDesligaSupG01,
	i_rSetPoint:= rSetPointTemperaturaSuperior[47],
	i_rProcessValue:= I_rTemperatura97,
	i_xManualMode:= ,
	i_rManualValue:= ,
	i_xAutoTune:= TEMP.xAutoTuneTemp97 OR xAutoTuneTempGeral,
	i_xHold:= ,
	i_xReset:= InterfaceHeat.xReset,
	i_stTemperatureControl:= stTemperatureControl[97],
	iq_etSelectParameterSetPID:= etSelectParameterSetPID[97],
	iq_stParameterSetsPID:= stParameterSetsPID[97],
	q_xActive=> ,
	q_xReady=> ,
	q_xError=> TEMP.xCrtlTemperatura[97],
	q_etResult=> TEMP.iCrtlTempStsTemp97,
	q_sResultMsg=> ,
	q_rAnalogOutput=> TEMP.rCrtlTempPotTemp97,
	q_xPwmOutput=> Q_xAquecimento97,
	q_xAutoTuneActive=> TEMP.xAutoTuneAtivoTemp97,
	q_etStatusAutoTune=> TEMP.iAutoTuneStsTemp97);

rPwmEntrada[97]:= TEMP.rCrtlTempPotTemp97*(rSetPorcentagemSuperior[47]/100);

PWM[97].i_stPara.tCyclTime:=T#10MS;
PWM[97].i_stPara.tPwmPeriod:=T#1000MS;
PWM[97](
	i_xEn:= 	xHabilitaBlocosControleSuperior,
	i_rIput:= 	rPwmEntrada[97],
	i_stPara:= 	,
	i_xErrRst:= xResetPid,
	q_xEn=> 	,
	q_xBusy=> 	,
	q_xPstv=> 	Q_xAquecimentoPwm97,
	q_xNgtv=> 	,
	q_xErr=> 	,
	q_uiErrId=> );

	// Controle Resistencia 98

SR_ControleTemperatura.FbCrtlAquecimento[98](
	i_xEnable:= InterfaceHeat.P_xHabTemp98 OR xLigaDesligaSupG02,
	i_rSetPoint:= rSetPointTemperaturaSuperior[48],
	i_rProcessValue:= I_rTemperatura98,
	i_xManualMode:= ,
	i_rManualValue:= ,
	i_xAutoTune:= TEMP.xAutoTuneTemp98 OR xAutoTuneTempGeral,
	i_xHold:= ,
	i_xReset:= InterfaceHeat.xReset,
	i_stTemperatureControl:= stTemperatureControl[98],
	iq_etSelectParameterSetPID:= etSelectParameterSetPID[98],
	iq_stParameterSetsPID:= stParameterSetsPID[98],
	q_xActive=> ,
	q_xReady=> ,
	q_xError=> TEMP.xCrtlTemperatura[98],
	q_etResult=> TEMP.iCrtlTempStsTemp98,
	q_sResultMsg=> ,
	q_rAnalogOutput=> TEMP.rCrtlTempPotTemp98,
	q_xPwmOutput=> Q_xAquecimento98,
	q_xAutoTuneActive=> TEMP.xAutoTuneAtivoTemp98,
	q_etStatusAutoTune=> TEMP.iAutoTuneStsTemp98);

	rPwmEntrada[98]:= TEMP.rCrtlTempPotTemp98*(rSetPorcentagemSuperior[48]/100);

PWM[98].i_stPara.tCyclTime:=T#10MS;
PWM[98].i_stPara.tPwmPeriod:=T#1000MS;
PWM[98](
	i_xEn:= 	xHabilitaBlocosControleSuperior,
	i_rIput:= 	rPwmEntrada[98],
	i_stPara:= 	,
	i_xErrRst:= xResetPid,
	q_xEn=> 	,
	q_xBusy=> 	,
	q_xPstv=> 	Q_xAquecimentoPwm98,
	q_xNgtv=> 	,
	q_xErr=> 	,
	q_uiErrId=> );

// Controle Resistencia 99

SR_ControleTemperatura.FbCrtlAquecimento[99](
	i_xEnable:= InterfaceHeat.P_xHabTemp99 OR xLigaDesligaSupG01,
	i_rSetPoint:= rSetPointTemperaturaSuperior[49],
	i_rProcessValue:= I_rTemperatura99,
	i_xManualMode:= ,
	i_rManualValue:= ,
	i_xAutoTune:= TEMP.xAutoTuneTemp99 OR xAutoTuneTempGeral,
	i_xHold:= ,
	i_xReset:= InterfaceHeat.xReset,
	i_stTemperatureControl:= stTemperatureControl[99],
	iq_etSelectParameterSetPID:= etSelectParameterSetPID[99],
	iq_stParameterSetsPID:= stParameterSetsPID[99],
	q_xActive=> ,
	q_xReady=> ,
	q_xError=> TEMP.xCrtlTemperatura[99],
	q_etResult=> TEMP.iCrtlTempStsTemp99,
	q_sResultMsg=> ,
	q_rAnalogOutput=> TEMP.rCrtlTempPotTemp99,
	q_xPwmOutput=> Q_xAquecimento99,
	q_xAutoTuneActive=> TEMP.xAutoTuneAtivoTemp99,
	q_etStatusAutoTune=> TEMP.iAutoTuneStsTemp99);

rPwmEntrada[99]:= TEMP.rCrtlTempPotTemp99*(rSetPorcentagemSuperior[49]/100);

PWM[99].i_stPara.tCyclTime:=T#10MS;
PWM[99].i_stPara.tPwmPeriod:=T#1000MS;
PWM[99](
	i_xEn:= 	xHabilitaBlocosControleSuperior,
	i_rIput:= 	rPwmEntrada[99],
	i_stPara:= 	,
	i_xErrRst:= xResetPid,
	q_xEn=> 	,
	q_xBusy=> 	,
	q_xPstv=> 	Q_xAquecimentoPwm99,
	q_xNgtv=> 	,
	q_xErr=> 	,
	q_uiErrId=> );

	// Controle Resistencia 100

SR_ControleTemperatura.FbCrtlAquecimento[100](
	i_xEnable:= InterfaceHeat.P_xHabTemp100 OR xLigaDesligaSupG02,
	i_rSetPoint:= rSetPointTemperaturaSuperior[50],
	i_rProcessValue:= I_rTemperatura100,
	i_xManualMode:= ,
	i_rManualValue:= ,
	i_xAutoTune:= TEMP.xAutoTuneTemp100 OR xAutoTuneTempGeral,
	i_xHold:= ,
	i_xReset:= InterfaceHeat.xReset,
	i_stTemperatureControl:= stTemperatureControl[100],
	iq_etSelectParameterSetPID:= etSelectParameterSetPID[100],
	iq_stParameterSetsPID:= stParameterSetsPID[100],
	q_xActive=> ,
	q_xReady=> ,
	q_xError=> TEMP.xCrtlTemperatura[100],
	q_etResult=> TEMP.iCrtlTempStsTemp100,
	q_sResultMsg=> ,
	q_rAnalogOutput=> TEMP.rCrtlTempPotTemp100,
	q_xPwmOutput=> Q_xAquecimento100,
	q_xAutoTuneActive=> TEMP.xAutoTuneAtivoTemp100,
	q_etStatusAutoTune=> TEMP.iAutoTuneStsTemp100);

rPwmEntrada[100]:= TEMP.rCrtlTempPotTemp100*(rSetPorcentagemSuperior[50]/100);

PWM[100].i_stPara.tCyclTime:=T#10MS;
PWM[100].i_stPara.tPwmPeriod:=T#1000MS;
PWM[100](
	i_xEn:= 	xHabilitaBlocosControleSuperior,
	i_rIput:= 	rPwmEntrada[100],
	i_stPara:= 	,
	i_xErrRst:= xResetPid,
	q_xEn=> 	,
	q_xBusy=> 	,
	q_xPstv=> 	Q_xAquecimentoPwm100,
	q_xNgtv=> 	,
	q_xErr=> 	,
	q_uiErrId=> );

//----------

	_30_AutoTunning();
